(* CODESYS project Валки.project
   CustomField01_name: CustomField01
   CustomField08_name: CustomField08
   CustomField06_name: CustomField06
   Title: ATV_IMC_Template
   CustomField09_name: CustomField09
   CustomField07_name: CustomField07
   CustomField05_name: CustomField05
   CustomField02_name: CustomField02
   Description: This template can be used for a correct interface with the local drive. the MANDATORY_AT_EACH_CYCLE program must be called like it is done in this application.
   CustomField04_name: CustomField04
   CustomField10_name: CustomField10
   Version: 0.0.0.0
   Company: Schneider Electric
   CustomField03_name: CustomField03

Project tree, tasks and I/O mapping:
  MyController : TM241CEC24T/U, Schneider Electric, order no. TM241CEC24T/U, version 4.0.3.8
    application Application
      task MAST (cyclic, interval 20 ms, priority 15, watchdog 100 ms x 1) calls MyPOU
      function HiddenPOU [ST]
      global variables GVL
      program MyPOU [LD]
      Symbols
    trace DeviceTrace (task ): 
    DI : Digital Inputs, Schneider Electric, version 4.0.3.8
        input  iwDI_IW0 : WORD  // IW0
        input  SB4_pusk : BOOL  // IW0.I8
        input  SB5_stop : BOOL  // IW0.I9
        input  SB6_pusk : BOOL  // IW0.I10
        input  SB7_stop : BOOL  // IW0.I11
        input  SB8_reset : BOOL  // IW0.I12
        input  ibDI_IB1 : BYTE  // IB1
    DQ : Digital Outputs, Schneider Electric, version 4.0.3.8
        output qwDQ_QW0 : WORD  // QW0
        output qbDQ_QB1 : BYTE  // QB1
    Counters : Counters, Schneider Electric, version 4.0.3.8
    Pulse_Generators : Pulse Generators, Schneider Electric, version 4.0.3.8
    Cartridge_1 : Cartridge, Schneider Electric, version 4.0.3.8
    IO_Bus : IO bus - TM3, Schneider Electric, version 4.0.3.8
      Module_3 : TM3DI32K, Schneider Electric, order no. TM3DI32K, version 1.0.1.2
          input  idwModule_3_ID0 : DWORD  // ID0
          input  QF_KM2 : BOOL  // ID0.I0
          input  QF_KM3 : BOOL  // ID0.I1
          input  QF_KM4 : BOOL  // ID0.I2
          input  QF_KM5 : BOOL  // ID0.I3
          input  QF_KM6 : BOOL  // ID0.I4
          input  QF_KM7 : BOOL  // ID0.I5
          input  QF_KM8 : BOOL  // ID0.I6
          input  QF_KM9 : BOOL  // ID0.I7
          input  QF_KM10 : BOOL  // ID0.I8
          input  QF_KM11 : BOOL  // ID0.I9
          input  Pusk_SB4 : BOOL  // ID0.I11
          input  Stop_SB5 : BOOL  // ID0.I12
          input  Pusk_SB6 : BOOL  // ID0.I13
          input  Stop_SB7 : BOOL  // ID0.I14
          input  Reset_SB8 : BOOL  // ID0.I15
          input  SQ1_merbrus : BOOL  // ID0.I16
          input  SQ2_ramAP : BOOL  // ID0.I17
          input  SQ3_ramDUN : BOOL  // ID0.I18
          input  SQ4_nalBrus : BOOL  // ID0.I19
          input  SQ5_PriKonDUN : BOOL  // ID0.I20
          input  SQ6_PriKonAP : BOOL  // ID0.I21
          input  SQ7_Tolk : BOOL  // ID0.I22
          input  SQ8_ : BOOL  // ID0.I23
          input  SQ9_OtKonAP : BOOL  // ID0.I24
          input  SQ10_OtKonDUN : BOOL  // ID0.I25
          input  SQ11_perKon : BOOL  // ID0.I26
          input  SQ12 : BOOL  // ID0.I27
          input  SQ13_Cistrun : BOOL  // ID0.I28
          input  FotoBor : BOOL  // ID0.I29
      Module_4 : TM3DQ16T/G, Schneider Electric, order no. TM3DQ16T/G, version 1.0.1.3
          output Kl1_KM2 : BOOL  // QB0.Q0
          output KL2_KM3 : BOOL  // QB0.Q1
          output KL3_KM4 : BOOL  // QB0.Q2
          output KL4_KM5 : BOOL  // QB0.Q3
          output KL5_KM6 : BOOL  // QB0.Q4
          output KL6_KM7 : BOOL  // QB0.Q5
          output KL7_KM8 : BOOL  // QB0.Q6
          output KL8_KM9 : BOOL  // QB0.Q7
          output KL9_KM10 : BOOL  // QB0.Q8
          output KL10_alarm : BOOL  // QB0.Q9
          output KL11_R : BOOL  // QB0.Q10
          output KL12_A : BOOL  // QB0.Q11
          output KL13_KM11 : BOOL  // QB0.Q12
          output KL14 : BOOL  // QB0.Q13
          output KL15 : BOOL  // QB0.Q14
          output KL16 : BOOL  // QB0.Q15
          unmapped channels: QB0
    COM_Bus : COM bus, Schneider Electric, version 4.0.3.8
    Ethernet_1 : Ethernet Network, Schneider Electric, version 4.0.3.8
        settings: IPAddress = [192, 168, 0, 150]; SubnetMask = [255, 255, 255, 0]; WebServer = TRUE; FTP Server = TRUE; SoMachine Protocol = TRUE; Modbus Server = TRUE; NetManage Protocol = TRUE; SNMP protocol = TRUE; Enable Routing = FALSE; WebVisu protocol = FALSE; DHCP Server Active = TRUE
      EthernetIP : EthernetIP, Schneider Electric, version 3.3.0.5
          unmapped channels: IW0, IW1, IW2, IW3, IW4, IW5, IW6, IW7, IW8, IW9, IW10, IW11, IW12, IW13, IW14, IW15, IW16, IW17, IW18, IW19, QW0, QW1, QW2, QW3, QW4, QW5, QW6, QW7, QW8, QW9, QW10, QW11, QW12, QW13, QW14, QW15, QW16, QW17, QW18, QW19
    Serial_Line_1 : Serial line, Schneider Electric, version 4.0.3.8
      SoMachine_Network_Manager : SoMachine-Network Manager, Schneider Electric, version 4.0.0.2
    Serial_Line_2 : Serial line, Schneider Electric, version 4.0.3.8
      SoMachine_Network_Manager_1 : SoMachine-Network Manager, Schneider Electric, version 4.0.0.2
    CAN_1 : CANopen bus, Schneider Electric, version 4.0.3.8
  HMIGTO4310 : HMIGTO4310, Schneider Electric, order no. HMIGTO4310, version 3.5.3.46
    HMI Application
    COM1
      SoMachine_Network_Manager1 : SoMachine-Network Manager, Schneider Electric, version 4.0.0.2
    COM2
      SoMachine_Network_Manager2 : SoMachine-Network Manager, Schneider Electric, version 4.0.0.2
    Ethernet
      SoMachine_Network_Manager3 : SoMachine-Network Manager, Schneider Electric, version 4.0.0.2
    USB
      SoMachine_Network_Manager4 : SoMachine-Network Manager, Schneider Electric, version 4.0.0.2
  FdtConnections : FDT Connections, Schneider Electric, version 1.0.0.2
    Modbus_Serial_Line_Manager : Modbus Serial Line Manager, Schneider Electric, version 2.2.0
  6c0f7fb6-600b-4c93-9262-20cdc603757e
*)

// MyController/Application/GVL
VAR_GLOBAL
	M_st: BOOL;
END_VAR

// MyController/Application/MyPOU
PROGRAM MyPOU
VAR
	m_SQ1: BOOL;
	TON_1: TON;
	mT_KM2: BOOL;
	TON_2: TON;
	m_KL2: BOOL;
	TON_3: TON;
	// бит работы подемного стола
	M_prictol: BOOL;
	TON_4: TON;
	M_TOLK: BOOL;
	TON_5: TON;
	Tim1: TIME;
	Tim2: TIME;
	Tim3: TIME;
	TON_6: TON;
	TON_7: TON;
	Tim4: TIME;
	TON_8: TON;
	Tim5: TIME;
	// фильтр работы датчика
	TON_9: TON;
	mSQ12: BOOL;
	TOF_11: TOF;
	Tim7: TIME;
	// время цикла работы подемного стола
	TON_10: TON;
	Tim6: TIME;
	mDunSQ12: BOOL;
	M_Kl1_KM2: BOOL;
	M_KL3_KM4: BOOL;
	M_KL4_KM5: BOOL;
	M_KL6_KM7: BOOL;
	M_KL9_KM10: BOOL;
	K_M_KL1_KM2: BOOL;
	mm_kl1_KM2: BOOL;
	K_M_KL3_KM4: BOOL;
	mm_KL3_KM4: BOOL;
	kl12a: BOOL;
	K_M_KL4_KM5: BOOL;
	mm_KL4_KM5: BOOL;
	K_M_KL6_KM7: BOOL;
	mm_KL6_KM7: BOOL;
	K_M_KL9_KM10: BOOL;
	mm_KL9_KM10: BOOL;
	K_M_KL2_KM3: BOOL;
	K_M_KL7_KM8: BOOL;
	M_K_KL8: BOOL;
	Tim10: TIME;
	M_KL5_KM6: BOOL;
	M_kl13: BOOL;
	TON_20: TON;
	In_tim1: INT := 2500;
	In_tim2: INT := 3100;
	In_tim3: INT := 2500;
	In_tim4: INT := 2500;
	In_tim5: INT := 2500;
	In_tim6: INT := 3000;
	In_tim7: INT := 3000;
	M_t3: BOOL;
	M_t4: BOOL;
	M_t5: BOOL;
	// приемный конвейер не в исходном положении
	Alarm_1: BOOL;
	// отдающий конвейер не в исходном положении
	Alarm_2: BOOL;
	M_pwr: BOOL;
END_VAR
VAR // added by the converter: edge detectors and wires of the graphical bodies
    _rt1, _rt2, _rt3, _rt4, _rt5, _rt6, _rt7, _rt8, _rt9, _rt10, _rt11, _rt12, _rt13, _rt14, _rt15, _rt16, _rt17, _rt18, _rt19, _rt20, _rt21, _rt22 : R_TRIG;
    _w1, _w2, _w3, _w4, _w5 : BOOL;
END_VAR

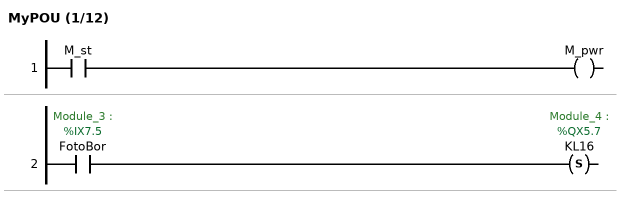
// NETWORK 1
M_pwr := M_st;

// NETWORK 2
//   FotoBor: Module_3 : | AT %IX7.5
//   KL16: Module_4 : | AT %QX5.7
KL16 S= FotoBor;

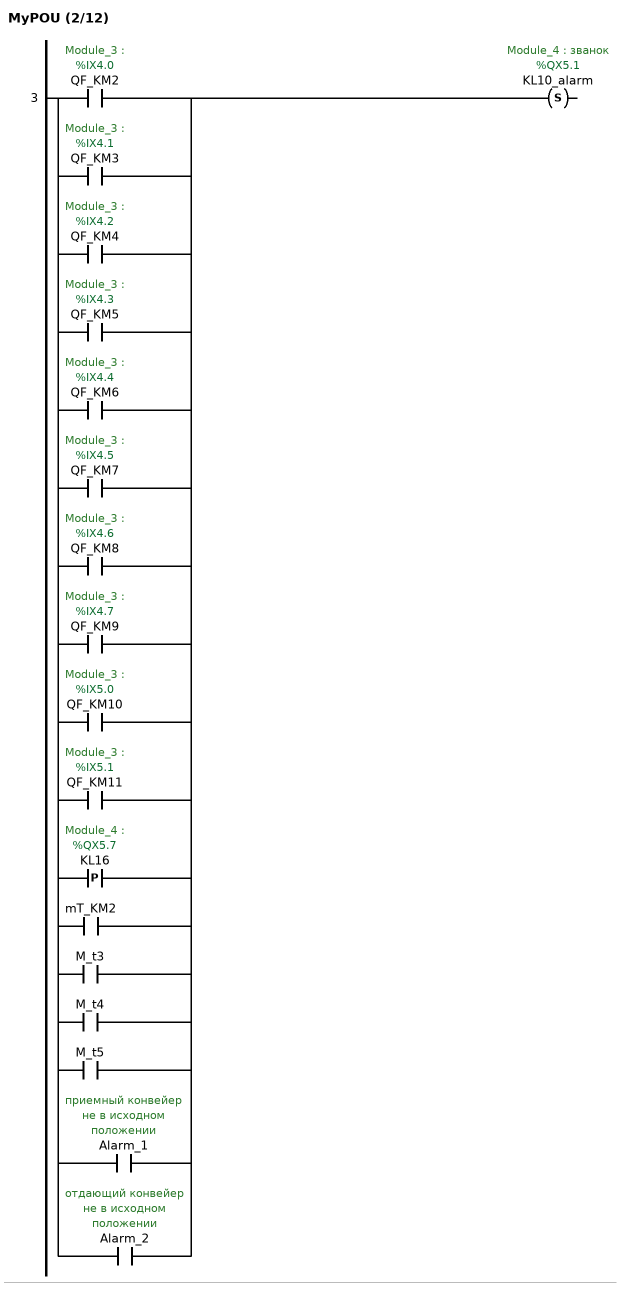
// NETWORK 3
//   QF_KM2: Module_3 : | AT %IX4.0
//   QF_KM3: Module_3 : | AT %IX4.1
//   QF_KM4: Module_3 : | AT %IX4.2
//   QF_KM5: Module_3 : | AT %IX4.3
//   QF_KM6: Module_3 : | AT %IX4.4
//   QF_KM7: Module_3 : | AT %IX4.5
//   QF_KM8: Module_3 : | AT %IX4.6
//   QF_KM9: Module_3 : | AT %IX4.7
//   QF_KM10: Module_3 : | AT %IX5.0
//   QF_KM11: Module_3 : | AT %IX5.1
//   KL16: Module_4 : | AT %QX5.7
//   Alarm_1: приемный конвейер не в исходном положении
//   Alarm_2: отдающий конвейер не в исходном положении
//   KL10_alarm: Module_4 : званок | AT %QX5.1
_rt1(CLK := KL16);
KL10_alarm S= QF_KM2 OR QF_KM3 OR QF_KM4 OR QF_KM5 OR QF_KM6 OR QF_KM7 OR QF_KM8 OR QF_KM9 OR QF_KM10 OR QF_KM11 OR _rt1.Q OR mT_KM2 OR M_t3 OR M_t4 OR M_t5 OR Alarm_1 OR Alarm_2;

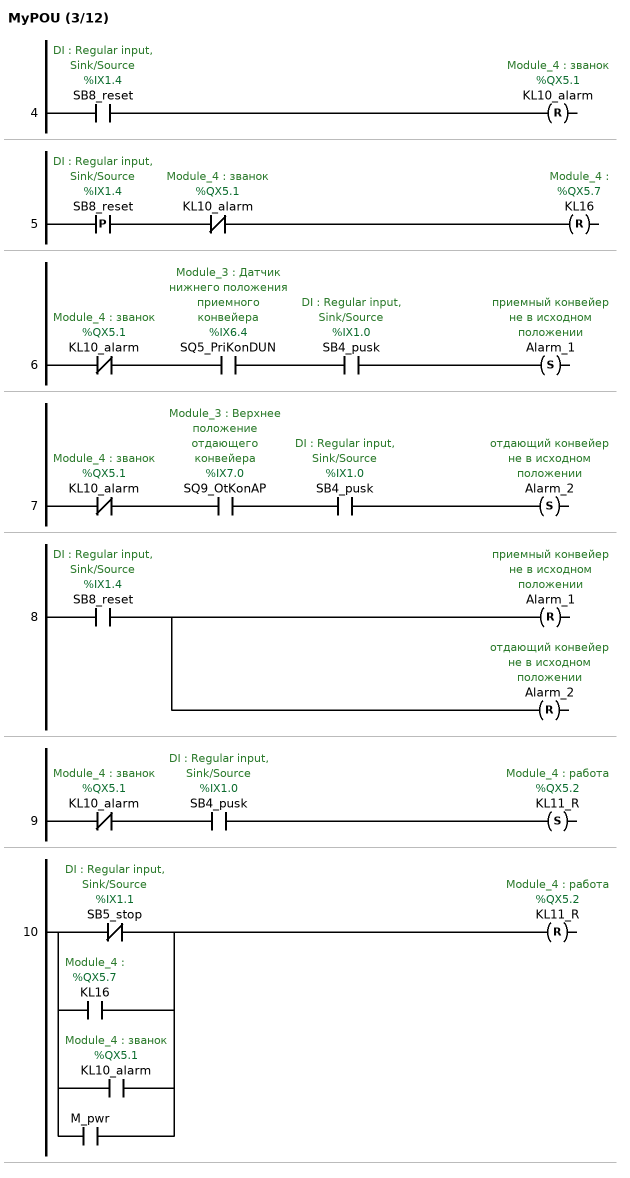
// NETWORK 4
//   SB8_reset: DI : Regular input, Sink/Source | AT %IX1.4
//   KL10_alarm: Module_4 : званок | AT %QX5.1
KL10_alarm R= SB8_reset;

// NETWORK 5
//   SB8_reset: DI : Regular input, Sink/Source | AT %IX1.4
//   KL10_alarm: Module_4 : званок | AT %QX5.1
//   KL16: Module_4 : | AT %QX5.7
_rt2(CLK := SB8_reset);
KL16 R= _rt2.Q AND NOT KL10_alarm;

// NETWORK 6
//   KL10_alarm: Module_4 : званок | AT %QX5.1
//   SQ5_PriKonDUN: Module_3 : Датчик нижнего положения приемного конвейера | AT %IX6.4
//   SB4_pusk: DI : Regular input, Sink/Source | AT %IX1.0
//   Alarm_1: приемный конвейер не в исходном положении
Alarm_1 S= NOT KL10_alarm AND SQ5_PriKonDUN AND SB4_pusk;

// NETWORK 7
//   KL10_alarm: Module_4 : званок | AT %QX5.1
//   SQ9_OtKonAP: Module_3 : Верхнее положение отдающего конвейера | AT %IX7.0
//   SB4_pusk: DI : Regular input, Sink/Source | AT %IX1.0
//   Alarm_2: отдающий конвейер не в исходном положении
Alarm_2 S= NOT KL10_alarm AND SQ9_OtKonAP AND SB4_pusk;

// NETWORK 8
//   SB8_reset: DI : Regular input, Sink/Source | AT %IX1.4
//   Alarm_1: приемный конвейер не в исходном положении
//   Alarm_2: отдающий конвейер не в исходном положении
Alarm_1 R= SB8_reset;
Alarm_2 R= SB8_reset;

// NETWORK 9
//   KL10_alarm: Module_4 : званок | AT %QX5.1
//   SB4_pusk: DI : Regular input, Sink/Source | AT %IX1.0
//   KL11_R: Module_4 : работа | AT %QX5.2
KL11_R S= NOT KL10_alarm AND SB4_pusk;

// NETWORK 10
//   SB5_stop: DI : Regular input, Sink/Source | AT %IX1.1
//   KL16: Module_4 : | AT %QX5.7
//   KL10_alarm: Module_4 : званок | AT %QX5.1
//   KL11_R: Module_4 : работа | AT %QX5.2
KL11_R R= NOT SB5_stop OR KL16 OR KL10_alarm OR M_pwr;

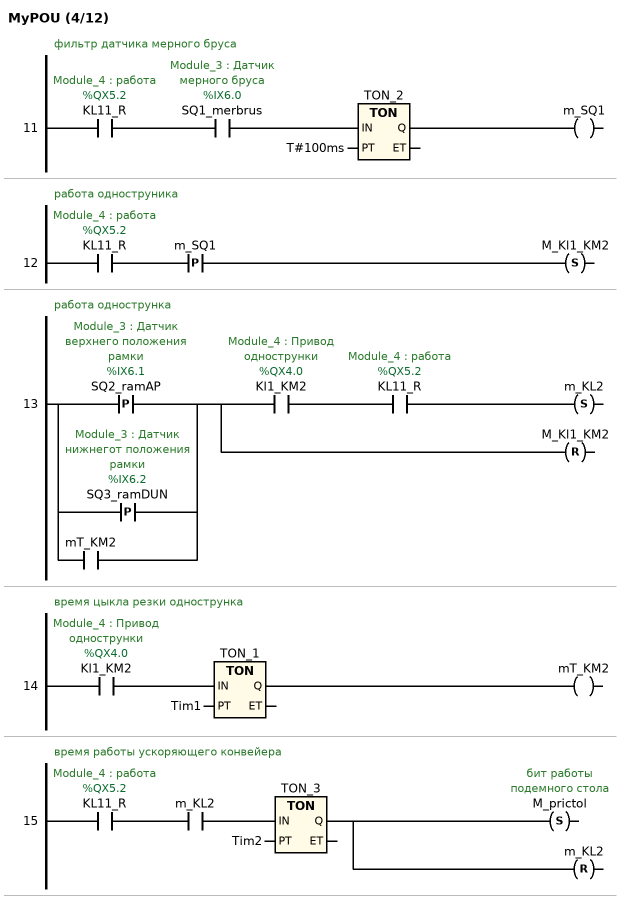
// NETWORK 11
// фильтр датчика мерного бруса
//   KL11_R: Module_4 : работа | AT %QX5.2
//   SQ1_merbrus: Module_3 : Датчик мерного бруса | AT %IX6.0
TON_2(IN := KL11_R AND SQ1_merbrus, PT := T#100ms); // TON
m_SQ1 := TON_2.Q;

// NETWORK 12
// работа одноструника
//   KL11_R: Module_4 : работа | AT %QX5.2
_rt3(CLK := m_SQ1);
M_Kl1_KM2 S= KL11_R AND _rt3.Q;

// NETWORK 13
// работа однострунка
//   SQ2_ramAP: Module_3 : Датчик верхнего положения рамки | AT %IX6.1
//   SQ3_ramDUN: Module_3 : Датчик нижнегот положения рамки | AT %IX6.2
//   Kl1_KM2: Module_4 : Привод однострунки | AT %QX4.0
//   KL11_R: Module_4 : работа | AT %QX5.2
_rt4(CLK := SQ2_ramAP);
_rt5(CLK := SQ3_ramDUN);
_w1 := _rt4.Q OR _rt5.Q OR mT_KM2;
m_KL2 S= _w1 AND Kl1_KM2 AND KL11_R;
M_Kl1_KM2 R= _w1;

// NETWORK 14
// время цыкла резки однострунка
//   Kl1_KM2: Module_4 : Привод однострунки | AT %QX4.0
TON_1(IN := Kl1_KM2, PT := Tim1); // TON
mT_KM2 := TON_1.Q;

// NETWORK 15
// время работы ускоряющего конвейера
//   KL11_R: Module_4 : работа | AT %QX5.2
//   M_prictol: бит работы подемного стола
TON_3(IN := KL11_R AND m_KL2, PT := Tim2); // TON
M_prictol S= TON_3.Q;
m_KL2 R= TON_3.Q;

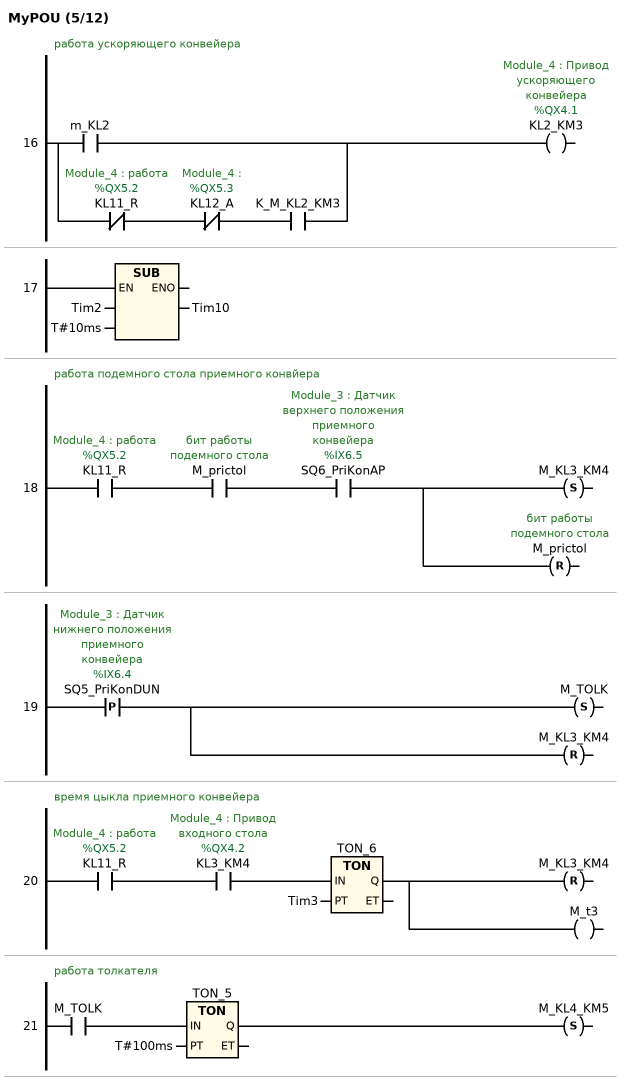
// NETWORK 16
// работа ускоряющего конвейера
//   KL11_R: Module_4 : работа | AT %QX5.2
//   KL12_A: Module_4 : | AT %QX5.3
//   KL2_KM3: Module_4 : Привод ускоряющего конвейера | AT %QX4.1
KL2_KM3 := m_KL2 OR NOT KL11_R AND NOT KL12_A AND K_M_KL2_KM3;

// NETWORK 17
Tim10 := Tim2 - T#10ms;

// NETWORK 18
// работа подемного стола приемного конвйера
//   KL11_R: Module_4 : работа | AT %QX5.2
//   M_prictol: бит работы подемного стола
//   SQ6_PriKonAP: Module_3 : Датчик верхнего положения приемного конвейера | AT %IX6.5
_w2 := KL11_R AND M_prictol AND SQ6_PriKonAP;
M_KL3_KM4 S= _w2;
M_prictol R= _w2;

// NETWORK 19
//   SQ5_PriKonDUN: Module_3 : Датчик нижнего положения приемного конвейера | AT %IX6.4
_rt6(CLK := SQ5_PriKonDUN);
M_TOLK S= _rt6.Q;
M_KL3_KM4 R= _rt6.Q;

// NETWORK 20
// время цыкла приемного конвейера
//   KL11_R: Module_4 : работа | AT %QX5.2
//   KL3_KM4: Module_4 : Привод входного стола | AT %QX4.2
TON_6(IN := KL11_R AND KL3_KM4, PT := Tim3); // TON
M_KL3_KM4 R= TON_6.Q;
M_t3 := TON_6.Q;

// NETWORK 21
// работа толкателя
TON_5(IN := M_TOLK, PT := T#100ms); // TON
M_KL4_KM5 S= TON_5.Q;

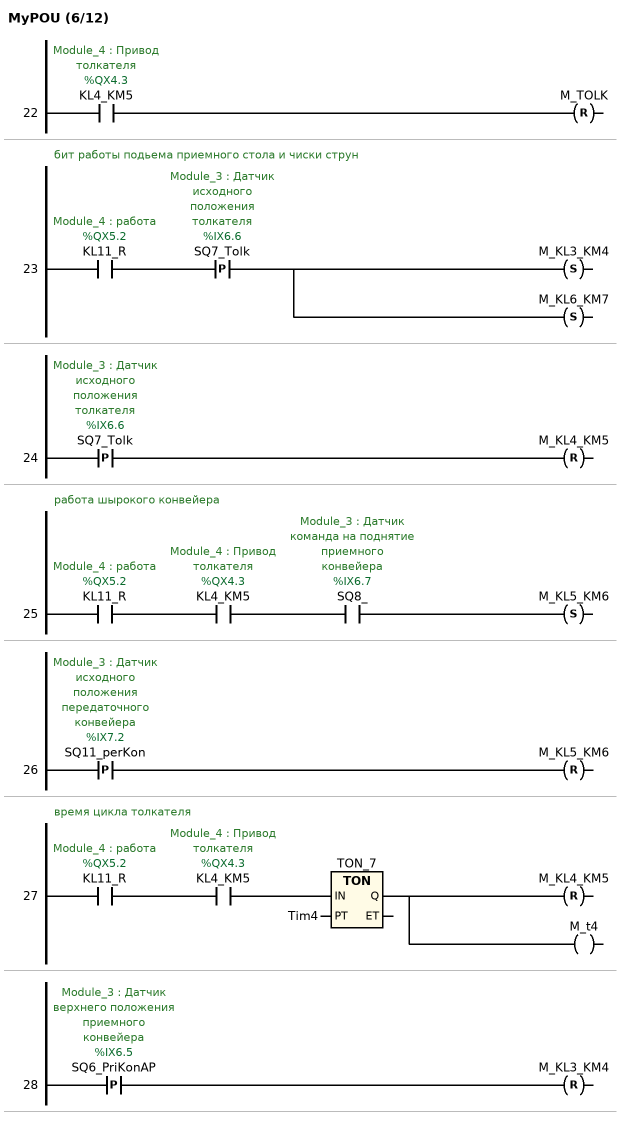
// NETWORK 22
//   KL4_KM5: Module_4 : Привод толкателя | AT %QX4.3
M_TOLK R= KL4_KM5;

// NETWORK 23
// бит работы подьема приемного стола и чиски струн
//   KL11_R: Module_4 : работа | AT %QX5.2
//   SQ7_Tolk: Module_3 : Датчик исходного положения толкателя | AT %IX6.6
_rt7(CLK := SQ7_Tolk);
_w3 := KL11_R AND _rt7.Q;
M_KL3_KM4 S= _w3;
M_KL6_KM7 S= _w3;

// NETWORK 24
//   SQ7_Tolk: Module_3 : Датчик исходного положения толкателя | AT %IX6.6
_rt8(CLK := SQ7_Tolk);
M_KL4_KM5 R= _rt8.Q;

// NETWORK 25
// работа шырокого конвейера
//   KL11_R: Module_4 : работа | AT %QX5.2
//   KL4_KM5: Module_4 : Привод толкателя | AT %QX4.3
//   SQ8_: Module_3 : Датчик команда на поднятие приемного конвейера | AT %IX6.7
M_KL5_KM6 S= KL11_R AND KL4_KM5 AND SQ8_;

// NETWORK 26
//   SQ11_perKon: Module_3 : Датчик исходного положения передаточного конвейера | AT %IX7.2
_rt9(CLK := SQ11_perKon);
M_KL5_KM6 R= _rt9.Q;

// NETWORK 27
// время цикла толкателя
//   KL11_R: Module_4 : работа | AT %QX5.2
//   KL4_KM5: Module_4 : Привод толкателя | AT %QX4.3
TON_7(IN := KL11_R AND KL4_KM5, PT := Tim4); // TON
M_KL4_KM5 R= TON_7.Q;
M_t4 := TON_7.Q;

// NETWORK 28
//   SQ6_PriKonAP: Module_3 : Датчик верхнего положения приемного конвейера | AT %IX6.5
_rt10(CLK := SQ6_PriKonAP);
M_KL3_KM4 R= _rt10.Q;

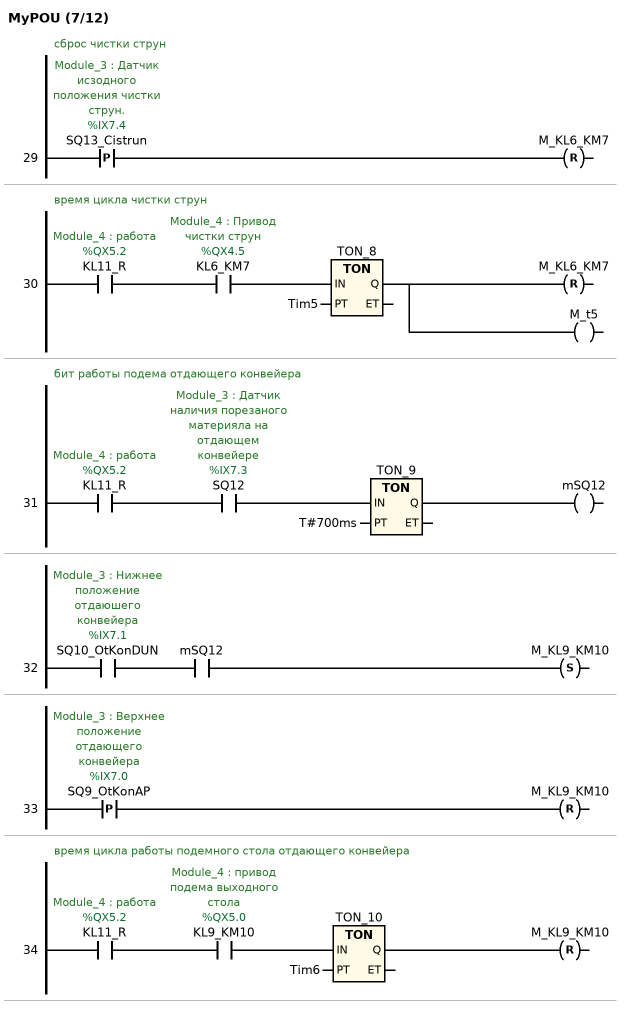
// NETWORK 29
// сброс чистки струн
//   SQ13_Cistrun: Module_3 : Датчик исзодного положения чистки струн. | AT %IX7.4
_rt11(CLK := SQ13_Cistrun);
M_KL6_KM7 R= _rt11.Q;

// NETWORK 30
// время цикла чистки струн
//   KL11_R: Module_4 : работа | AT %QX5.2
//   KL6_KM7: Module_4 : Привод чистки струн | AT %QX4.5
TON_8(IN := KL11_R AND KL6_KM7, PT := Tim5); // TON
M_KL6_KM7 R= TON_8.Q;
M_t5 := TON_8.Q;

// NETWORK 31
// бит работы подема отдающего конвейера
//   TON_9: фильтр работы датчика
//   KL11_R: Module_4 : работа | AT %QX5.2
//   SQ12: Module_3 : Датчик наличия порезаного материяла на отдающем конвейере | AT %IX7.3
TON_9(IN := KL11_R AND SQ12, PT := T#700ms); // TON
mSQ12 := TON_9.Q;

// NETWORK 32
//   SQ10_OtKonDUN: Module_3 : Нижнее положение отдаюшего конвейера | AT %IX7.1
M_KL9_KM10 S= SQ10_OtKonDUN AND mSQ12;

// NETWORK 33
//   SQ9_OtKonAP: Module_3 : Верхнее положение отдающего конвейера | AT %IX7.0
_rt12(CLK := SQ9_OtKonAP);
M_KL9_KM10 R= _rt12.Q;

// NETWORK 34
// время цикла работы подемного стола отдающего конвейера
//   TON_10: время цикла работы подемного стола
//   KL11_R: Module_4 : работа | AT %QX5.2
//   KL9_KM10: Module_4 : привод подема выходного стола | AT %QX5.0
TON_10(IN := KL11_R AND KL9_KM10, PT := Tim6); // TON
M_KL9_KM10 R= TON_10.Q;

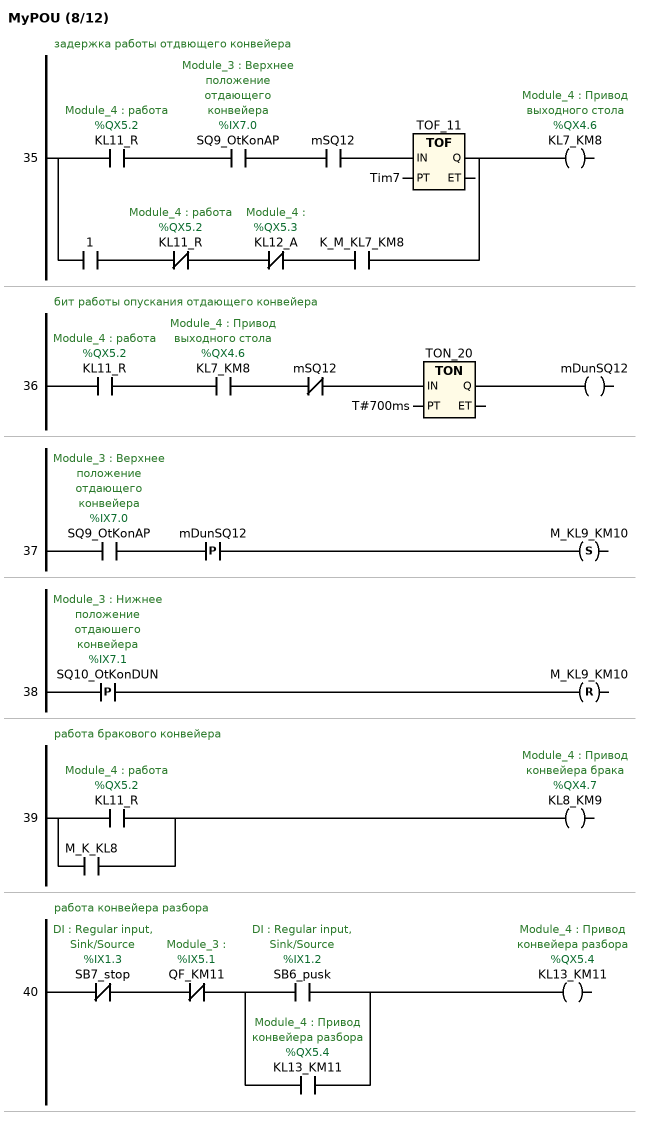
// NETWORK 35
// задержка работы отдвющего конвейера
//   KL11_R: Module_4 : работа | AT %QX5.2
//   SQ9_OtKonAP: Module_3 : Верхнее положение отдающего конвейера | AT %IX7.0
//   KL12_A: Module_4 : | AT %QX5.3
//   KL7_KM8: Module_4 : Привод выходного стола | AT %QX4.6
TOF_11(IN := KL11_R AND SQ9_OtKonAP AND mSQ12, PT := Tim7); // TOF
KL7_KM8 := TOF_11.Q OR 1 AND NOT KL11_R AND NOT KL12_A AND K_M_KL7_KM8;

// NETWORK 36
// бит работы опускания отдающего конвейера
//   KL11_R: Module_4 : работа | AT %QX5.2
//   KL7_KM8: Module_4 : Привод выходного стола | AT %QX4.6
TON_20(IN := KL11_R AND KL7_KM8 AND NOT mSQ12, PT := T#700ms); // TON
mDunSQ12 := TON_20.Q;

// NETWORK 37
//   SQ9_OtKonAP: Module_3 : Верхнее положение отдающего конвейера | AT %IX7.0
_rt13(CLK := mDunSQ12);
M_KL9_KM10 S= SQ9_OtKonAP AND _rt13.Q;

// NETWORK 38
//   SQ10_OtKonDUN: Module_3 : Нижнее положение отдаюшего конвейера | AT %IX7.1
_rt14(CLK := SQ10_OtKonDUN);
M_KL9_KM10 R= _rt14.Q;

// NETWORK 39
// работа бракового конвейера
//   KL11_R: Module_4 : работа | AT %QX5.2
//   KL8_KM9: Module_4 : Привод конвейера брака | AT %QX4.7
KL8_KM9 := KL11_R OR M_K_KL8;

// NETWORK 40
// работа конвейера разбора
//   SB7_stop: DI : Regular input, Sink/Source | AT %IX1.3
//   QF_KM11: Module_3 : | AT %IX5.1
//   SB6_pusk: DI : Regular input, Sink/Source | AT %IX1.2
//   KL13_KM11: Module_4 : Привод конвейера разбора | AT %QX5.4
KL13_KM11 := NOT SB7_stop AND NOT QF_KM11 AND (SB6_pusk OR KL13_KM11);

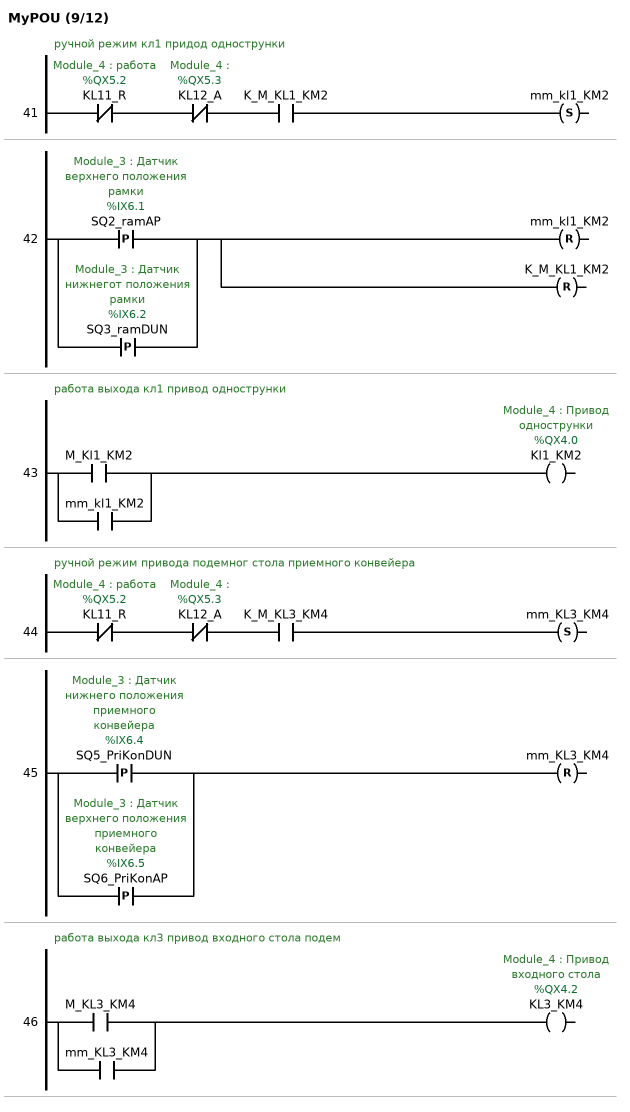
// NETWORK 41
// ручной режим кл1 придод однострунки
//   KL11_R: Module_4 : работа | AT %QX5.2
//   KL12_A: Module_4 : | AT %QX5.3
mm_kl1_KM2 S= NOT KL11_R AND NOT KL12_A AND K_M_KL1_KM2;

// NETWORK 42
//   SQ2_ramAP: Module_3 : Датчик верхнего положения рамки | AT %IX6.1
//   SQ3_ramDUN: Module_3 : Датчик нижнегот положения рамки | AT %IX6.2
_rt15(CLK := SQ2_ramAP);
_rt16(CLK := SQ3_ramDUN);
_w4 := _rt15.Q OR _rt16.Q;
mm_kl1_KM2 R= _w4;
K_M_KL1_KM2 R= _w4;

// NETWORK 43
// работа выхода кл1 привод однострунки
//   Kl1_KM2: Module_4 : Привод однострунки | AT %QX4.0
Kl1_KM2 := M_Kl1_KM2 OR mm_kl1_KM2;

// NETWORK 44
// ручной режим привода подемног стола приемного конвейера
//   KL11_R: Module_4 : работа | AT %QX5.2
//   KL12_A: Module_4 : | AT %QX5.3
mm_KL3_KM4 S= NOT KL11_R AND NOT KL12_A AND K_M_KL3_KM4;

// NETWORK 45
//   SQ5_PriKonDUN: Module_3 : Датчик нижнего положения приемного конвейера | AT %IX6.4
//   SQ6_PriKonAP: Module_3 : Датчик верхнего положения приемного конвейера | AT %IX6.5
_rt17(CLK := SQ5_PriKonDUN);
_rt18(CLK := SQ6_PriKonAP);
mm_KL3_KM4 R= _rt17.Q OR _rt18.Q;

// NETWORK 46
// работа выхода кл3 привод входного стола подем
//   KL3_KM4: Module_4 : Привод входного стола | AT %QX4.2
KL3_KM4 := M_KL3_KM4 OR mm_KL3_KM4;

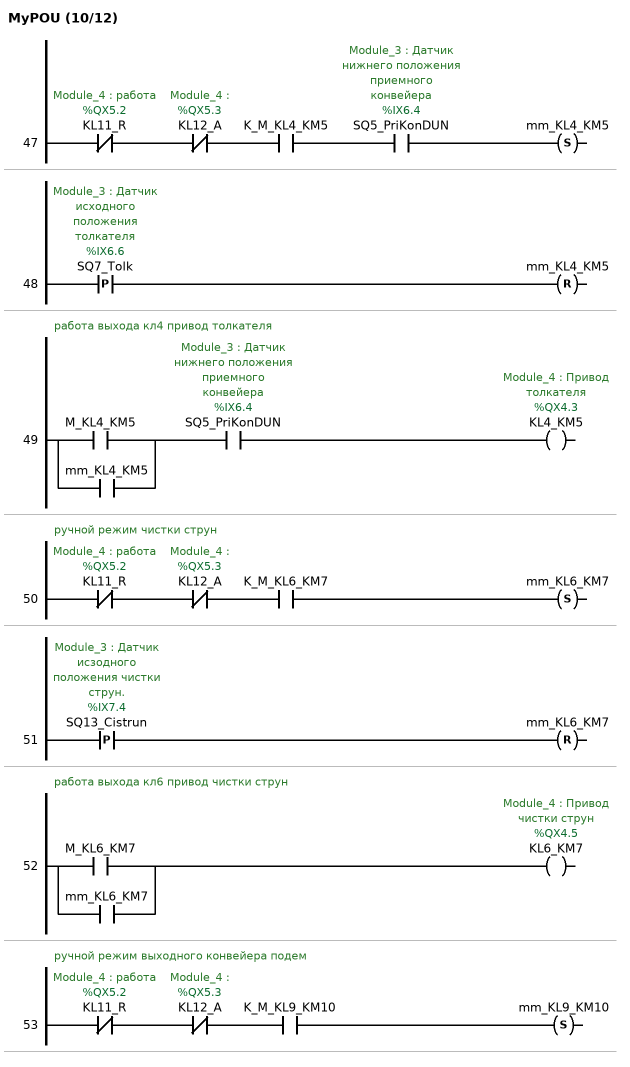
// NETWORK 47
//   KL11_R: Module_4 : работа | AT %QX5.2
//   KL12_A: Module_4 : | AT %QX5.3
//   SQ5_PriKonDUN: Module_3 : Датчик нижнего положения приемного конвейера | AT %IX6.4
mm_KL4_KM5 S= NOT KL11_R AND NOT KL12_A AND K_M_KL4_KM5 AND SQ5_PriKonDUN;

// NETWORK 48
//   SQ7_Tolk: Module_3 : Датчик исходного положения толкателя | AT %IX6.6
_rt19(CLK := SQ7_Tolk);
mm_KL4_KM5 R= _rt19.Q;

// NETWORK 49
// работа выхода кл4 привод толкателя
//   SQ5_PriKonDUN: Module_3 : Датчик нижнего положения приемного конвейера | AT %IX6.4
//   KL4_KM5: Module_4 : Привод толкателя | AT %QX4.3
KL4_KM5 := (M_KL4_KM5 OR mm_KL4_KM5) AND SQ5_PriKonDUN;

// NETWORK 50
// ручной режим чистки струн
//   KL11_R: Module_4 : работа | AT %QX5.2
//   KL12_A: Module_4 : | AT %QX5.3
mm_KL6_KM7 S= NOT KL11_R AND NOT KL12_A AND K_M_KL6_KM7;

// NETWORK 51
//   SQ13_Cistrun: Module_3 : Датчик исзодного положения чистки струн. | AT %IX7.4
_rt20(CLK := SQ13_Cistrun);
mm_KL6_KM7 R= _rt20.Q;

// NETWORK 52
// работа выхода кл6 привод чистки струн
//   KL6_KM7: Module_4 : Привод чистки струн | AT %QX4.5
KL6_KM7 := M_KL6_KM7 OR mm_KL6_KM7;

// NETWORK 53
// ручной режим выходного конвейера подем
//   KL11_R: Module_4 : работа | AT %QX5.2
//   KL12_A: Module_4 : | AT %QX5.3
mm_KL9_KM10 S= NOT KL11_R AND NOT KL12_A AND K_M_KL9_KM10;

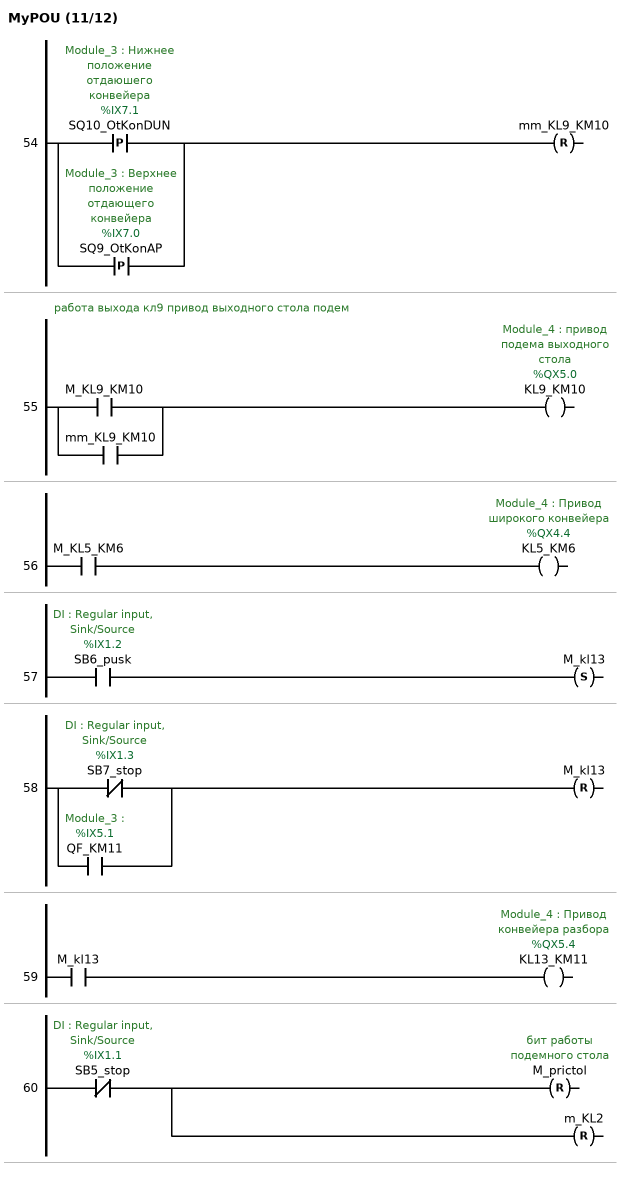
// NETWORK 54
//   SQ10_OtKonDUN: Module_3 : Нижнее положение отдаюшего конвейера | AT %IX7.1
//   SQ9_OtKonAP: Module_3 : Верхнее положение отдающего конвейера | AT %IX7.0
_rt21(CLK := SQ10_OtKonDUN);
_rt22(CLK := SQ9_OtKonAP);
mm_KL9_KM10 R= _rt21.Q OR _rt22.Q;

// NETWORK 55
// работа выхода кл9 привод выходного стола подем
//   KL9_KM10: Module_4 : привод подема выходного стола | AT %QX5.0
KL9_KM10 := M_KL9_KM10 OR mm_KL9_KM10;

// NETWORK 56
//   KL5_KM6: Module_4 : Привод широкого конвейера | AT %QX4.4
KL5_KM6 := M_KL5_KM6;

// NETWORK 57
//   SB6_pusk: DI : Regular input, Sink/Source | AT %IX1.2
M_kl13 S= SB6_pusk;

// NETWORK 58
//   SB7_stop: DI : Regular input, Sink/Source | AT %IX1.3
//   QF_KM11: Module_3 : | AT %IX5.1
M_kl13 R= NOT SB7_stop OR QF_KM11;

// NETWORK 59
//   KL13_KM11: Module_4 : Привод конвейера разбора | AT %QX5.4
KL13_KM11 := M_kl13;

// NETWORK 60
//   SB5_stop: DI : Regular input, Sink/Source | AT %IX1.1
//   M_prictol: бит работы подемного стола
_w5 := NOT SB5_stop;
M_prictol R= _w5;
m_KL2 R= _w5;

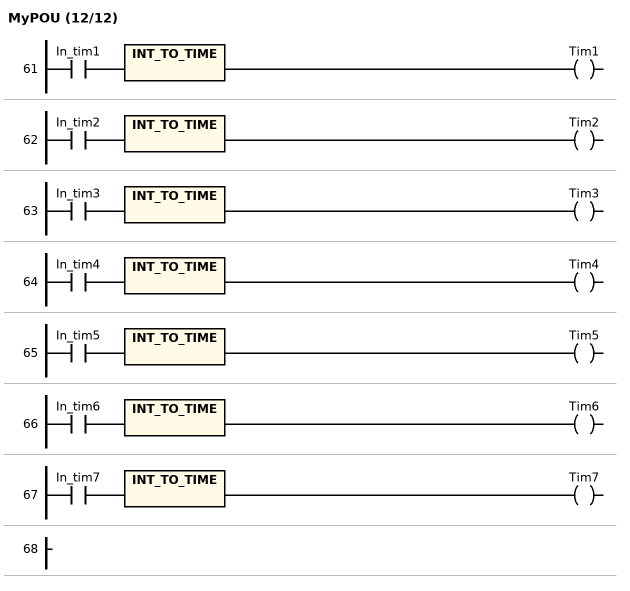
// NETWORK 61
Tim1 := INT_TO_TIME(In_tim1);

// NETWORK 62
Tim2 := INT_TO_TIME(In_tim2);

// NETWORK 63
Tim3 := INT_TO_TIME(In_tim3);

// NETWORK 64
Tim4 := INT_TO_TIME(In_tim4);

// NETWORK 65
Tim5 := INT_TO_TIME(In_tim5);

// NETWORK 66
Tim6 := INT_TO_TIME(In_tim6);

// NETWORK 67
Tim7 := INT_TO_TIME(In_tim7);

// NETWORK 68

END_PROGRAM

// MyController/Application/HiddenPOU
FUNCTION HiddenPOU : BOOL

VAR_INPUT
	pHiddenFunc: POINTER TO WORD;
END_VAR
VAR
	pRead: POINTER TO BYTE;
	pWrite: POINTER TO BYTE;
END_VAR

pRead := pHiddenFunc + 400;
pWrite := pHiddenFunc + 4400;
HiddenPOU := TRUE;

END_FUNCTION
